Staubli VAL3: setAlarm.pgx

program setAlarm(num x_nNum)
begin
  switch x_nNum
    case 0
      dAlarm[0]=true
      dAlarm[1]=false
      dAlarm[2]=false
      dAlarm[3]=false
      dAlarm[4]=false
      dAlarm[5]=false
      dAlarm[6]=false
      dAlarm[7]=false
      delay(0.35)
      dAlarm[0]=false
      dAlarm[1]=false
      dAlarm[2]=false
      dAlarm[3]=false
      dAlarm[4]=false
      dAlarm[5]=false
      dAlarm[6]=false
      dAlarm[7]=false
    break
    case 1
      dAlarm[0]=false
      dAlarm[1]=true
      dAlarm[2]=false
      dAlarm[3]=false
      dAlarm[4]=false
      dAlarm[5]=false
      dAlarm[6]=false
      dAlarm[7]=false
      delay(0.35)
      dAlarm[0]=false
      dAlarm[1]=false
      dAlarm[2]=false
      dAlarm[3]=false
      dAlarm[4]=false
      dAlarm[5]=false
      dAlarm[6]=false
      dAlarm[7]=false
    break
    case 2
      dAlarm[0]=false
      dAlarm[1]=false
      dAlarm[2]=true
      dAlarm[3]=false
      dAlarm[4]=false
      dAlarm[5]=false
      dAlarm[6]=false
      dAlarm[7]=false
      delay(0.35)
      dAlarm[0]=false
      dAlarm[1]=false
      dAlarm[2]=false
      dAlarm[3]=false
      dAlarm[4]=false
      dAlarm[5]=false
      dAlarm[6]=false
      dAlarm[7]=false
    break
    case 3
      dAlarm[0]=false
      dAlarm[1]=false
      dAlarm[2]=true
      dAlarm[3]=false
      dAlarm[4]=false
      dAlarm[5]=false
      dAlarm[6]=false
      dAlarm[7]=false
      delay(0.35)
      dAlarm[0]=false
      dAlarm[1]=false
      dAlarm[2]=false
      dAlarm[3]=false
      dAlarm[4]=false
      dAlarm[5]=false
      dAlarm[6]=false
      dAlarm[7]=false
    break
    case 4
      dAlarm[0]=false
      dAlarm[1]=false
      dAlarm[2]=false
      dAlarm[3]=false
      dAlarm[4]=true
      dAlarm[5]=false
      dAlarm[6]=false
      dAlarm[7]=false
      delay(0.35)
      dAlarm[0]=false
      dAlarm[1]=false
      dAlarm[2]=false
      dAlarm[3]=false
      dAlarm[4]=false
      dAlarm[5]=false
      dAlarm[6]=false
      dAlarm[7]=false
    break
    case 5
      dAlarm[0]=false
      dAlarm[1]=false
      dAlarm[2]=false
      dAlarm[3]=false
      dAlarm[4]=false
      dAlarm[5]=true
      dAlarm[6]=false
      dAlarm[7]=false
      delay(0.35)
      dAlarm[0]=false
      dAlarm[1]=false
      dAlarm[2]=false
      dAlarm[3]=false
      dAlarm[4]=false
      dAlarm[5]=false
      dAlarm[6]=false
      dAlarm[7]=false
    break
    case 6
      dAlarm[0]=false
      dAlarm[1]=false
      dAlarm[2]=false
      dAlarm[3]=false
      dAlarm[4]=false
      dAlarm[5]=false
      dAlarm[6]=true
      dAlarm[7]=false
      delay(0.35)
      dAlarm[0]=false
      dAlarm[1]=false
      dAlarm[2]=false
      dAlarm[3]=false
      dAlarm[4]=false
      dAlarm[5]=false
      dAlarm[6]=false
      dAlarm[7]=false
    break
    case 7
      dAlarm[0]=false
      dAlarm[1]=false
      dAlarm[2]=false
      dAlarm[3]=false
      dAlarm[4]=false
      dAlarm[5]=false
      dAlarm[6]=false
      dAlarm[7]=true
      delay(0.35)
      dAlarm[0]=false
      dAlarm[1]=false
      dAlarm[2]=false
      dAlarm[3]=false
      dAlarm[4]=false
      dAlarm[5]=false
      dAlarm[6]=false
      dAlarm[7]=false
    break
    default
      dAlarm[0]=false
      dAlarm[1]=false
      dAlarm[2]=false
      dAlarm[3]=false
      dAlarm[4]=false
      dAlarm[5]=false
      dAlarm[6]=false
      dAlarm[7]=false
    break
  endSwitch
end
